Fanuc KAREL source: kd00066.KL

-- PROVISIONAL review KL for V1013-1; original PC SHA256 f552a78fefc2f204b6e836a043f313f069470d94ef43eb2051f0200addef16e4
-- Incomplete behavior may be omitted. Consult companion uncertainty JSON. Do not deploy.
PROGRAM KD00066
%NOLOCKGROUP
VAR
  I : INTEGER
  J : INTEGER
  B : BOOLEAN
  R : REAL
  S : STRING[80]
BEGIN
  -- UNRESOLVED_PC offsets 5-17; opcodes 9D,81,18,9D,1B,9D,12,13,04
  -- UNRESOLVED_PC offsets 22-26; opcodes 7F
END KD00066
